PROGRAM MAIN
VAR_INPUT
	execute : BOOL;
	manualMode : BOOL;
END_VAR
VAR_OUTPUT
	robotLeft, robotRight : Robot;
	
	skidLeft, skidRight : MaterialStorage;
	stagingTableLeft, stagingTableRight : WoodBunkTable;
	magazineLeft, magazineRight : MaterialStorage;
	
	strapper : StrapMachine;
	
	insertionLeft, insertionRight : PneumaticInsertion;	
	insertionBottom : TeknicEIP;
	topSuction : ARRAY[1..3] OF SuctionPad;
	leftSuction, rightSuction : ARRAY[1..4] OF SuctionPad;
	bottomSuction : ARRAY[1..2] OF SuctionPad;
	
	toolStorageLeft : A21ToolStorage;
	toolStorageRight : A21ToolStorage;
	
	stagingTemplateLeft, stagingTemplateRight : WoodBunkTable;
END_VAR
VAR
	robotLeftOutputs, robotRightOutputs : ARRAY[1..50] OF INT;
	demoPairWB : PositionMaterials;
	demoPairCIP : PositionMaterials;
	demoHeight : REAL := 600; //600mm, 60cm
	
	sectionID : SectionEnum := SectionEnum.WOOD_BUNK;
	
	step : (IDLE, STAGING, LOAD_CIP, LOAD_WB, PUSH, STRAP, RELEASE, COMPLETE := 1050);
	ready : BOOL;
	
	loadSet : INT;
	loadStepLeft, loadStepRight : INT;
	
	stageSet : INT;	
	stageStepLeft, stageStepRight : INT;
	iStagingSlotLeft, iStagingSlotRight : INT;
END_VAR
VAR CONSTANT
	//COMPLETE : INT := 1050;
END_VAR

demoPairWB.position := 0;
demoPairWB.top := 'WDW20';
demoPairWB.left := 'WDS14';
demoPairWB.right := 'WDS14';
demoPairWB.bottom := 'WDB20';

demoPairCIP.position := 0;
demoPairCIP.top := 'CIP54';
demoPairCIP.bottom := 'CIP18';

setup();
hardwareLadder();

IF NOT ready THEN
	ready :=
		insertionLeft.homingSequence() AND
		insertionRight.homingSequence() AND
		insertionBottom.homingSequence();
END_IF


CASE step OF
	IDLE:
		IF execute THEN
			execute := FALSE;
			step := LOAD_CIP;
		END_IF
	
	LOAD_CIP:
		IF loadCIP(pair:= demoPairWB) THEN
			IF manualMode AND_THEN NOT execute THEN
				RETURN;
			END_IF
		
			step := STAGING;
		END_IF
		
	STAGING:
		IF stage() THEN
			IF manualMode AND_THEN NOT execute THEN
				RETURN;
			END_IF
			
			step := LOAD_CIP;
		END_IF
		
	LOAD_WB:
		IF loadWB(pair := demoPairWB) THEN
			IF manualMode AND_THEN NOT execute THEN
				RETURN;
			END_IF
		
			step := STRAP;
		END_IF
		
	PUSH:
		insertionBottom.traverse(direction := FALSE);
		IF NOT insertionLeft.alignTarget(demoHeight/2) OR insertionRight.alignTarget(demoHeight/2) THEN
			RETURN;
		END_IF
		
		insertionBottom.traverse(direction := FALSE);
		insertionLeft.press();
		insertionRight.press();
		
		IF insertionBottom.contact AND insertionLeft.contact AND insertionRight.contact THEN
			step := STRAP;
		END_IF
		
	STRAP:
		IF strapper.ready OR (NOT strapper.busy AND NOT strapper.error) THEN
			strapper.strap();
		END_IF
		
		IF strapper.done THEN
			IF manualMode AND_THEN NOT execute THEN
				RETURN;
			END_IF
			
			step := RELEASE;
		END_IF
		
	RELEASE: //release command
		MEMSET(ADR(topSuction), 0, SIZEOF(topSuction));
		MEMSET(ADR(leftSuction), 0, SIZEOF(leftSuction));
		MEMSET(ADR(rightSuction), 0, SIZEOF(rightSuction));
		MEMSET(ADR(bottomSuction), 0, SIZEOF(bottomSuction));
		
		IF NOT insertionLeft.home THEN
			insertionLeft.alignTarget(0);
			insertionLeft.release();
		END_IF
		
		IF NOT insertionRight.home THEN
			insertionRight.alignTarget(0);
			insertionRight.release();
		END_IF
		
		IF insertionLeft.home AND insertionRight.home THEN
			IF manualMode AND_THEN NOT execute THEN
				RETURN;
			END_IF
			
			step := COMPLETE;
		END_IF
	
	COMPLETE:
		//reset everything
		step := IDLE;
		
END_CASE

METHOD changeRobotsEOAT : BOOL
VAR_INPUT
	targetTool : SectionEnum;
END_VAR
IF robotLeft.tool <> sectionID THEN
	MEMSET(ADR(robotLeftOutputs), 0, SIZEOF(robotLeftOutputs));
	robotLeftOutputs[1] := A21.TOOL_CHANGE_CHIPBOARD;
	robotLeft.setParamsAndWait(robotLeftOutputs);
END_IF

IF robotRight.tool <> sectionID THEN
	MEMSET(ADR(robotRightOutputs), 0, SIZEOF(robotRightOutputs));
	robotRightOutputs[1] := A21.TOOL_CHANGE_CHIPBOARD;
	robotRight.setParamsAndWait(robotRightOutputs);
END_IF

changeRobotsEOAT := robotLeft.tool = sectionID AND robotRight.tool = sectionID;
END_METHOD

METHOD PROTECTED createStagingTemplate : BOOL
VAR
	remainingMaterial : STRING;
	splitMaterial : STRING;
	
	i : INT;
END_VAR
stagingTemplateLeft.autofill(demoPairWB.top);
stagingTemplateLeft.autofill(demoPairWB.left);

stagingTemplateRight.autofill(demoPairWB.right);
stagingTemplateRight.autofill(demoPairWB.bottom);

createStagingTemplate := TRUE;

(*
FOR i:=0 TO GVL.maxPairs BY 1 DO //iterate through all pairs and autofill the template
	//LEFT TABLE
	remainingMaterial := materialsArr[i].top;
	WHILE FIND(remainingMaterial, '_') > 0 DO //until no underscore found
		splitCombinedMaterials(remainingMaterial, splitMaterial);
		stagingTemplateLeft.autofill(splitMaterial);
	END_WHILE
	stagingTemplateLeft.autofill(remainingMaterial);
	
	remainingMaterial := materialsArr[i].left;
	WHILE FIND(remainingMaterial, '_') > 0 DO
		splitCombinedMaterials(remainingMaterial, splitMaterial);
		stagingTemplateLeft.autofill(splitMaterial);
	END_WHILE
	stagingTemplateLeft.autofill(remainingMaterial);
	
	//RIGHT TABLE
	remainingMaterial := materialsArr[i].right;
	WHILE FIND(remainingMaterial, '_') > 0 DO
		splitCombinedMaterials(remainingMaterial, splitMaterial);
		stagingTemplateRight.autofill(splitMaterial);
	END_WHILE
	stagingTemplateRight.autofill(remainingMaterial);
	
	remainingMaterial := materialsArr[i].bottom;
	WHILE FIND(remainingMaterial, '_') > 0 DO
		splitCombinedMaterials(remainingMaterial, splitMaterial);
		stagingTemplateRight.autofill(splitMaterial);
	END_WHILE
	stagingTemplateRight.autofill(remainingMaterial);
END_FOR
createStagingTemplate := TRUE;
*)
END_METHOD

METHOD hardwareCall : BOOL
robotLeft();
robotRight();

skidLeft();
skidRight();

stagingTableLeft();
stagingTableRight();

magazineLeft();
magazineRight();

strapper();

insertionLeft();
insertionRight();
insertionBottom();

stagingTemplateLeft();
stagingTemplateRight();
END_METHOD

METHOD hardwareLadder : BOOL
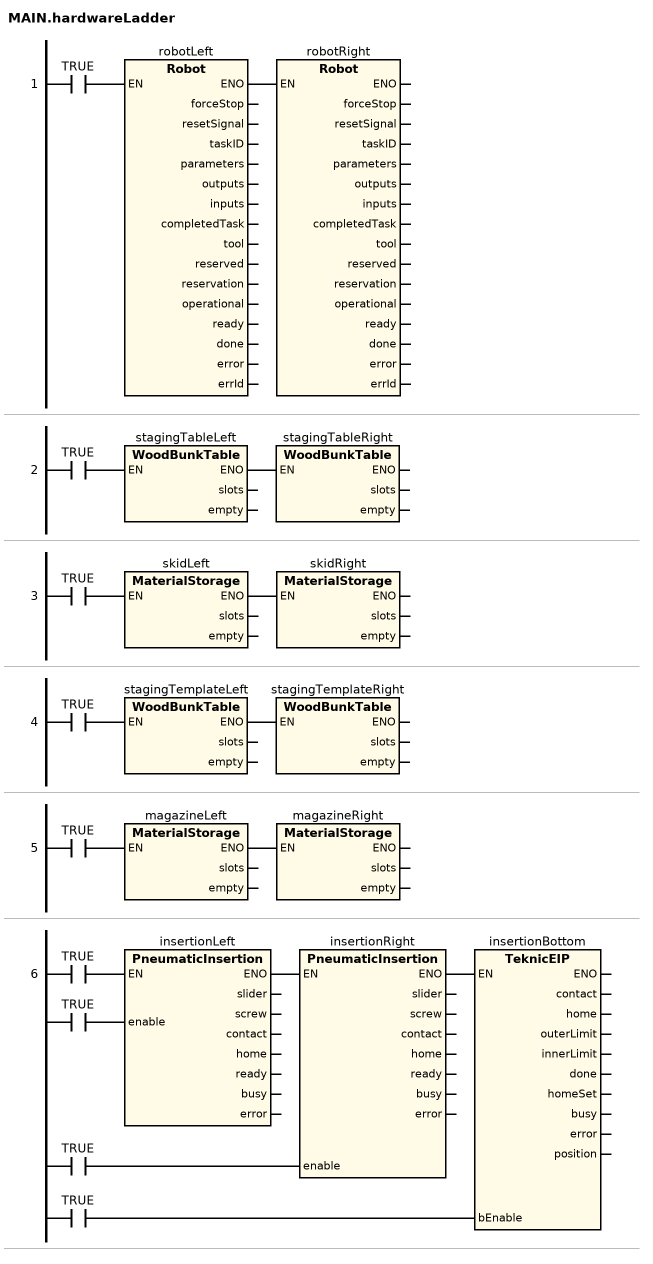
// NETWORK 1
robotLeft(); // Robot
robotRight(); // Robot

// NETWORK 2
stagingTableLeft(); // WoodBunkTable
stagingTableRight(); // WoodBunkTable

// NETWORK 3
skidLeft(); // MaterialStorage
skidRight(); // MaterialStorage

// NETWORK 4
stagingTemplateLeft(); // WoodBunkTable
stagingTemplateRight(); // WoodBunkTable

// NETWORK 5
magazineLeft(); // MaterialStorage
magazineRight(); // MaterialStorage

// NETWORK 6
insertionLeft(enable := TRUE); // PneumaticInsertion
insertionRight(enable := TRUE); // PneumaticInsertion
insertionBottom(bEnable := TRUE); // TeknicEIP
END_METHOD

METHOD loadCIP : BOOL
VAR_INPUT
	pair : REFERENCE TO PositionMaterials;
END_VAR
VAR_OUTPUT
	error : BOOL;
END_VAR
IF NOT robotLeft.operational AND NOT robotLeft.operational THEN
	error := TRUE;
	RETURN;
END_IF

IF NOT (robotLeft.reserve(SectionEnum.CHIPBOARD) AND robotRight.reserve(SectionEnum.CHIPBOARD)) THEN
	RETURN;
END_IF

IF NOT (robotLeft.tool = SectionEnum.CHIPBOARD AND robotRight.tool = SectionEnum.CHIPBOARD) THEN //robots have wrong tool
	changeRobotsEOAT(SectionEnum.CHIPBOARD); //wait for robots to finish changing tools
	RETURN;
END_IF


CASE loadSet OF
	0: //demo only - only top chipboard loaded by left robot
		IF 
			loadingSequenceCIP(
				actingRobot:= robotLeft, 
				robotOutputs:= robotLeftOutputs, 
				storage:= skidLeft, 
				loadStep:= loadStepLeft, 
				surfaceID:= Surface.TOP,
				material:= pair.top, 
				fail=> )
		THEN
			loadStepLeft := loadStepRight := 0;
			loadSet := 10;
		END_IF
		
	10: //recovery
		IF robotLeft.operational AND NOT robotRight.operational THEN //left ok, right fail
			IF
				loadingSequenceCIP(
					actingRobot:= robotLeft, 
					robotOutputs:= robotLeftOutputs, 
					storage:= skidLeft, 
					loadStep:= loadStepLeft, 
					surfaceID:= Surface.BOTTOM,
					material:= pair.top, 
					fail=> ) //load bottom with left robot
			THEN
				step := COMPLETE;
			END_IF
			
		ELSIF NOT robotLeft.operational AND robotRight.operational THEN //left fail, right ok
			IF
				loadingSequenceCIP(
					actingRobot:= robotRight, 
					robotOutputs:= robotRightOutputs, 
					storage:= skidRight, 
					loadStep:= loadStepRight, 
					surfaceID:= Surface.TOP,
					material:= pair.bottom, 
					fail=> ) //load top with right robot
			THEN
				step := COMPLETE;
			END_IF
			
		END_IF
		
	COMPLETE:
		loadSet := 0;
		loadStepLeft := loadStepRight := 0;
		
		robotLeft.release(sectionID);
		robotRight.release(sectionID);
		
		loadCIP := TRUE;
END_CASE
END_METHOD

METHOD loadingSequenceCIP : BOOL
VAR_IN_OUT
	actingRobot : Robot;
	robotOutputs : ARRAY[1..50] OF INT;
	storage : MaterialStorage;
	loadStep : INT;
END_VAR
VAR_INPUT
	surfaceID : Surface;
	material : STRING;
END_VAR
VAR_OUTPUT
	fail : BOOL;
END_VAR
VAR
	slot : INT;
END_VAR
IF material = '' THEN
	loadingSequenceCIP := TRUE;
	RETURN;
END_IF

CASE loadStep OF
	0:
		IF NOT storage.findSlot(materialID := material, atSlot => slot) THEN
			fail := TRUE;
			RETURN;
		END_IF
		
		MEMSET(ADR(robotOutputs), 0, SIZEOF(robotOutputs));
		robotOutputs[1] := A21.GET_CHIPBOARD_FROM_SKID;
		robotOutputs[2] := slot;
		
		CASE surfaceID OF
			Surface.TOP:
				IF actingRobot.setParamsAndWait(robotOutputs) THEN
					loadStep := 10;
				END_IF
				
			Surface.BOTTOM:
				//lower conveyor
				IF actingRobot.setParamsAndWait(robotOutputs) (*AND conveyor lowered*) THEN
					loadStep := 10;
				END_IF
			
		END_CASE
		
	10:
		MEMSET(ADR(robotOutputs), 0, SIZEOF(robotOutputs));
		CASE surfaceID OF
			Surface.TOP: 					robotOutputs[1] := A21.PLACE_CHIPBOARD_TO_TOP;
			Surface.BOTTOM: 				robotOutputs[1] := A21.PLACE_CHIPBOARD_TO_BOTTOM;
		END_CASE
		robotOutputs[2] := slot;
		
		IF actingRobot.setParamsAndWait(robotOutputs) THEN
			loadStep := 10;
		END_IF
		
	COMPLETE:
		actingRobot.release(sectionID);
		loadingSequenceCIP := TRUE;
		
END_CASE
END_METHOD

METHOD loadingSequenceWB : BOOL
VAR_IN_OUT
	actingRobot : Robot;
	robotOutputs : ARRAY[1..50] OF INT;
	stagingTable : WoodBunkTable;
	suctions : ARRAY[*] OF SuctionPad;
	loadStep : INT;
END_VAR
VAR_INPUT
	surfaceID : Surface;
	material : STRING;
END_VAR
VAR_OUTPUT
	fail : BOOL;
END_VAR
VAR
	slot : INT;
	i : DINT;
END_VAR
IF material = '' THEN
	loadingSequenceWB := TRUE;
	RETURN;
END_IF

CASE loadStep OF
	0:
		IF NOT stagingTable.findSlot(materialID := material, atSlot => slot) THEN
			fail := TRUE;
			RETURN;
		END_IF
		
		MEMSET(ADR(robotOutputs), 0, SIZEOF(robotOutputs));
		CASE surfaceID OF
			Surface.TOP: 					robotOutputs[1] := A21.LOAD_BUNK_TO_TOP;
			Surface.LEFT, Surface.RIGHT: 	robotOutputs[1] := A21.LOAD_BUNK_TO_SIDE;
			Surface.BOTTOM: 				robotOutputs[1] := A21.LOAD_BUNK_TO_BOTTOM;
		END_CASE
		robotOutputs[2] := slot;
		
		IF actingRobot.setParamsAndWait(robotOutputs) THEN
			loadStep := COMPLETE;
		END_IF
		
	COMPLETE:
		FOR i:=LOWER_BOUND(suctions, 1) TO UPPER_BOUND(suctions, 1) BY 1 DO
			suctions[i].enable := TRUE;
		END_FOR
		
		loadingSequenceWB := TRUE;
		
END_CASE
END_METHOD

METHOD PROTECTED loadWB : BOOL
VAR_INPUT
	pair : REFERENCE TO PositionMaterials;
END_VAR
VAR_OUTPUT
	error : BOOL;
END_VAR
IF NOT robotLeft.operational OR NOT robotLeft.operational THEN
	error := TRUE;
	RETURN;
END_IF

IF NOT (robotLeft.reserve(SectionEnum.WOOD_BUNK) AND robotRight.reserve(SectionEnum.WOOD_BUNK)) THEN
	RETURN;
END_IF

IF NOT (robotLeft.tool = SectionEnum.WOOD_BUNK AND robotRight.tool = SectionEnum.WOOD_BUNK) THEN //robots have wrong tool
	changeRobotsEOAT(SectionEnum.WOOD_BUNK); //wait for robots to finish changing tools
	RETURN;
END_IF

CASE loadSet OF
	0: //top and bottom
		IF 
			loadingSequenceWB(
				actingRobot:= robotLeft, 
				robotOutputs:= robotLeftOutputs, 
				stagingTable:= stagingTableLeft, 
				loadStep:= loadStepLeft, 
				suctions:= topSuction,
				surfaceID:= Surface.TOP, 
				material:= pair.top, 
				fail=> )
			AND
			loadingSequenceWB(
				actingRobot:= robotRight, 
				robotOutputs:= robotRightOutputs, 
				stagingTable:= stagingTableRight, 
				loadStep:= loadStepRight, 
				suctions:= bottomSuction,
				surfaceID:= Surface.BOTTOM, 
				material:= pair.bottom, 
				fail=> )
		THEN
			loadStepLeft := loadStepRight := 0;
			loadSet := 10;
		END_IF
		
	10: //sides
		IF
			loadingSequenceWB(
				actingRobot:= robotLeft, 
				robotOutputs:= robotLeftOutputs, 
				stagingTable:= stagingTableLeft, 
				loadStep:= loadStepLeft, 
				suctions:= leftSuction,
				surfaceID:= Surface.LEFT, 
				material:= pair.left, 
				fail=> )
			AND
			loadingSequenceWB(
				actingRobot:= robotRight, 
				robotOutputs:= robotRightOutputs, 
				stagingTable:= stagingTableRight, 
				loadStep:= loadStepRight, 
				suctions:= rightSuction,
				surfaceID:= Surface.RIGHT, 
				material:= pair.right, 
				fail=> )
		THEN
			loadStepLeft := loadStepRight := 0;
			loadSet := COMPLETE;
		END_IF
		
	COMPLETE:
		loadSet := 0;
		loadStepLeft := loadStepRight := 0;
		
		robotLeft.release(sectionID);
		robotRight.release(sectionID);
		
		loadWB := TRUE;
END_CASE
END_METHOD

METHOD PRIVATE setup : BOOL
VAR
	iWoodBunkSlot : WoodBunk := 1;
	iChipboardSlot : Chipboard := 1;
	
	slotsArr : ARRAY[1..GVL.maxQueue] OF STRING;
	
	i : INT;
END_VAR
FOR iWoodBunkSlot:=1 TO WoodBunk.size-1 BY 1 DO
	slotsArr[iWoodBunkSlot] := TO_STRING(iWoodBunkSlot);
END_FOR
magazineLeft.setupSlots(slotsArr);
magazineRight.setupSlots(slotsArr);

FOR iChipboardSlot:=1 TO Chipboard.size-1 BY 1 DO
	slotsArr[iChipboardSlot] := TO_STRING(iChipboardSlot);
END_FOR
skidLeft.setupSlots(slotsArr);
skidRight.setupSlots(slotsArr);


insertionLeft.enable := insertionRight.enable := insertionBottom.bEnable := TRUE;

setup := TRUE;
END_METHOD

METHOD stage : BOOL
//robot reservation needs to be constantly checked so it is not in the state machine
IF NOT (robotLeft.reserve(sectionID) AND robotRight.reserve(sectionID)) THEN
	RETURN;
END_IF

IF NOT (robotLeft.tool = SectionEnum.WOOD_BUNK AND robotRight.tool = SectionEnum.WOOD_BUNK) THEN //robots have wrong tool
	changeRobotsEOAT(SectionEnum.WOOD_BUNK); //wait for robots to finish changing tools
	RETURN;
END_IF

CASE stageSet OF
	0: //create staging template
		IF createStagingTemplate() THEN
			step := 10;
		END_IF
	
	10: //staging sequence
		IF
			stagingSequence(
				template:= stagingTemplateLeft, 
				magazine:= magazineLeft, 
				table:= stagingTableLeft, 
				actingStagingSlot:= iStagingSlotLeft,
				actingRobot:= robotLeft, 
				robotOutputs:= robotLeftOutputs,
				actingStep:= stageStepLeft, 
				fail=> )
				
			AND
			stagingSequence(
				template:= stagingTemplateRight, 
				magazine:= magazineRight, 
				table:= stagingTableRight, 
				actingStagingSlot:= iStagingSlotRight,
				actingRobot:= robotRight, 
				robotOutputs:= robotRightOutputs,
				actingStep:= stageStepRight, 
				fail=> )
		THEN
			stageStepLeft := stageStepRight := 0;
			iStagingSlotLeft := iStagingSlotRight := 0;
			
			stageSet := COMPLETE;
		END_IF
		
	COMPLETE:
		stageSet := 0;
		stageStepLeft := stageStepRight := 0;
		
		robotLeft.release(sectionID);
		robotRight.release(sectionID);
		
		stage := TRUE;
		
END_CASE
END_METHOD

METHOD stageLeft : BOOL
VAR_IN_OUT
	template : WoodBunkTable;
	magazine : MaterialStorage;
	table : WoodBunkTable;
	actingStagingSlot : INT;
	actingRobot : Robot;
	robotOutputs : ARRAY[1..50] OF INT;
	actingStep : INT;
END_VAR
VAR_OUTPUT
	fail : BOOL;
END_VAR
VAR
	finished : BOOL;
	
	slot : INT;
	templateArr : POINTER TO STRING;
	//iSlot : REFERENCE TO INT; 
END_VAR
VAR CONSTANT
	WIP : INT := 0;
	PASSED : INT := 1;
	FAILED : INT := 2;
END_VAR
(*
IF table.isFull() OR actingStagingSlot > 10 THEN
	stageLeft := TRUE;
	RETURN;
END_IF

templateArr := template.getSlotsAsArray();

//follow the template as is
IF NOT magazine.findSlot(materialID:= templateArr[actingStagingSlot], atSlot => slot) THEN
	fail := TRUE;
	RETURN;
END_IF

IF actingStep > 0 THEN
	finished := actingRobot.setParamsAndWait(robotOutputs);
END_IF

CASE actingStep OF		
	0:
		IF actingRobot.inputs[5].10 THEN //in position for inspection
			robotOutputs[4] := PASSED;
			actingStep := 30;
		END_IF
		
	COMPLETE:
		IF finished THEN
			actingStep := 0;
		END_IF
END_CASE
*)
END_METHOD

METHOD stageRight : BOOL
VAR_IN_OUT
	template : WoodBunkTable;
	magazine : MaterialStorage;
	table : WoodBunkTable;
	actingStagingSlot : INT;
	actingRobot : Robot;
	actingStep : INT;
END_VAR
VAR_INPUT
	camera : INT;
END_VAR
VAR_OUTPUT
	fail : BOOL;
END_VAR
VAR
	finished : BOOL;
	robotOutputs : POINTER TO INT;
	
	slot : INT;
	templateArr : POINTER TO STRING;
	
END_VAR
(*
IF table.isFull() OR actingStagingSlot > 10 THEN
	stageRight := TRUE;
	RETURN;
END_IF

templateArr := template.getSlotsAsArray();

//follow the template as is
IF NOT magazine.findSlot(materialID:= templateArr[actingStagingSlot], atSlot => slot) THEN
	fail := TRUE;
	RETURN;
END_IF

IF actingStep > 0 THEN
	finished := actingRobot.setCommandAndWait(A21.STAGE_BUNK, slot, actingStagingSlot, 0);
END_IF

CASE actingStep OF
	0: //command
		IF actingRobot.inputs[5].10 THEN
			actingStep := 10;
		END_IF
		
	10: //send inspection data
		tempInspectionSuite.frame.MaterialID := templateArr[actingStagingSlot];
		tempInspectionSuite.frame.CheckFor := 'ORIENTATION';
		tempInspectionSuite.frame.CameraNumber := camera;
	
		CreateJsonDocumentAuto(
			visionFrameData:= tempInspectionSuite.frame, 
			jsonDocument=> tempInspectionSuite.json);
		
		MEMCPY( //data = json
			ADR(tempInspectionSuite.data), 
			ADR(tempInspectionSuite.json), 
			MIN( SIZEOF(tempInspectionSuite.data), SIZEOF(tempInspectionSuite.json) ));
			
		TcpServer1Vision.queue(tempInspectionSuite.data);
		
		actingStep := 20;
	
	20: //fetch inspection data and parse
		actingRobot.setCommandAndWait(A21.STAGE_BUNK, slot, actingStagingSlot, 0);
		robotOutputs[11] := 0;
		
		IF NOT FrameIsValid(actingFrame) THEN
			RETURN;
		END_IF
		
		IF actingFrame.SuccessFlag = 1 THEN
			robotOutputs[11] := 1;
		ELSE
			robotOutputs[11] := 2;
		END_IF
		step := 30;
		
	30: //finish command
		IF finished THEN
			IF actingFrame.SuccessFlag = 1 THEN
				actingStagingSlot := actingStagingSlot + 1;
			END_IF
			
			actingStep := 0; //stage next
		END_IF
		
END_CASE
*)
END_METHOD

METHOD stagingSequence : BOOL
VAR_IN_OUT
	template : WoodBunkTable;
	magazine : MaterialStorage;
	table : WoodBunkTable;
	actingStagingSlot : INT;
	actingRobot : Robot;
	robotOutputs : ARRAY[1..50] OF INT;
	actingStep : INT;
END_VAR
VAR_OUTPUT
	fail : BOOL;
END_VAR
VAR
	finished : BOOL;
	slot : INT;
	templateArr : POINTER TO STRING;
END_VAR
VAR CONSTANT
	WIP : INT := 0;
	PASSED : INT := 1;
	FAILED : INT := 2;
END_VAR
IF
	table.isFull() OR actingStagingSlot > 10 OR //table full
	MEMCMP(ADR(table.slots), templateArr, SIZEOF(table.slots)) = 0 //table matches template
	//MEMCMP(table.getSlotsAsArray(), templateArr, SIZEOF(templateArr)) = 0
THEN
	stagingSequence := TRUE;
	RETURN;
END_IF

templateArr := ADR(template.slots);

//follow the template as is
IF NOT magazine.findSlot(materialID:= templateArr[actingStagingSlot], atSlot => slot) THEN
	fail := TRUE;
	RETURN;
END_IF

IF actingStep > 0 THEN
	finished := actingRobot.setParamsAndWait(robotOutputs);
END_IF

CASE actingStep OF		
	0:
		IF actingRobot.inputs[5].10 THEN //in position for inspection
			robotOutputs[4] := PASSED;
			actingStep := 30;
		END_IF
		
	30:
		IF finished THEN
			actingStep := COMPLETE;
		END_IF
		
	COMPLETE:
		MEMSET(ADR(robotOutputs), 0, SIZEOF(robotOutputs));
		actingStagingSlot := actingStagingSlot + 1;
		//stagingSequence := TRUE;
END_CASE
END_METHOD

END_PROGRAM

(* stored: Version 1.1.0.1, ProductVersion 3.1.4024.11
   POU MAIN: Id {f31366c8-7465-4414-aaf4-fb935af985c5}, SpecialFunc None
   Folder Loading: Id {6998e9bf-e2b9-4fd9-897f-fda9aa3bdaab}
   Folder Staging: Id {df129403-abf4-453c-addd-f6dd4ee3c4b1}
   Method changeRobotsEOAT: Id {71a414a6-260d-4ed7-9b91-4169239414f1}
   Method createStagingTemplate: Id {7fe7b744-7294-4b6c-b036-1426eaceb21a}
   Method hardwareCall: Id {ae27e4e1-f18c-46c6-a88d-05763e2b1498}
   Method hardwareLadder: Id {9403ad4a-57c3-4db6-915e-1dd4d905aad6}
   Method loadCIP: Id {4d48d146-da99-4898-b32c-d988fd277adc}
   Method loadingSequenceCIP: Id {dab34edb-3da5-4404-8c49-3d0bd468a2d2}
   Method loadingSequenceWB: Id {ec5e74a4-d8f7-4a78-89ca-cd705faa47d2}
   Method loadWB: Id {b6e713a8-dc8d-419f-844e-f7d0d4b22dfa}
   Method setup: Id {0ba728b9-6522-4c82-81e3-44efce8fc95c}
   Method stage: Id {413ca9c3-a808-4782-b740-b91ebf3df60f}
   Method stageLeft: Id {3b8fe327-e7eb-4f4b-b513-70d48c9a8543}
   Method stageRight: Id {27442b6e-36aa-485b-84ba-8788912b7a2c}
   Method stagingSequence: Id {a405d3c7-f8a4-4bcd-a99a-948da7c9242e} *)
